PROGRAM ModbusRTU
VAR
	fbEpcMb: ModbusRtuMaster_KL6x22B;
	wQty: WORD;
	wMbAddr: WORD;
	wData: ARRAY[1..10] OF WORD;
	bRead: BOOL;
	fbRTrigRead: R_TRIG;
END_VAR

fbRTrigRead(CLK:=bRead, Q=>);

IF fbRTrigRead.Q THEN
	wQty := 10;
	wMbAddr := 20;
END_IF

fbEpcMb.ReadRegs(
	UnitID:= 10, 
	Quantity:= wQty, 
	MBAddr:= wMbAddr, 
	cbLength:= SIZEOF(wData), 
	pMemoryAddr:= ADR(wData), 
	Execute:= fbRTrigRead.Q, 
	Timeout:= T#2S, 
	BUSY=> , 
	Error=> , 
	ErrorId=> , 
	cbRead=> );

END_PROGRAM

(* stored: Version 1.1.0.1, ProductVersion 3.1.4024.12
   POU ModbusRTU: Id {fb1103b6-429f-46ca-a932-ab687a9dc31f}, SpecialFunc None *)
